TYPE U_MOVE_DATA :
UNION
  stData              : ARRAY[1..MAX_MOVER] OF ST_MOVE_DATA;

  byData    AT %Q*    : ARRAY[1..MAX_MOVER] OF
                        ARRAY[1..SIZEOF(ST_MOVE_DATA)] OF BYTE;
END_UNION
END_TYPE

(* stored: Version 1.1.0.1
   DUT U_MOVE_DATA: Id {dfe7bcb9-0978-4c0c-8db9-967e7dca0322} *)
